# EPICS autosave request: ipApp/Db/ADAM_4015_chan_settings.req
$(P)$(R):rtd$(C).DESC
$(P)$(R):rtd$(C).SCAN
$(P)$(R):temp$(C).DESC
$(P)$(R):unit$(C).VAL
